INTERFACE I_TransformLRealValue EXTENDS I_Base

METHOD Transform : LREAL
VAR_INPUT
	Value	: LREAL;
	Reverse : BOOL := FALSE;
END_VAR
END_METHOD

END_INTERFACE

(* stored: Version 1.1.0.1, ProductVersion 3.1.4026.18
   Itf I_TransformLRealValue: Id {22ad0c43-610b-42b6-abb5-16b5dfbb58be}
   Method Transform: Id {17374df7-51e7-45a1-87c2-a56139abbfda} *)
